// TIA Portal V20 export
TYPE "typeCmInterfaceSoftCam"
// stored: Access Published, Namespace Unit1.Em5
   STRUCT
      ngAndManualInput : "Unit1.Em5.typeCminterfaceSoftCamManualInput";
      magazine : "Unit1.Em5.typeCminterfaceSoftCamMagazine";
   END_STRUCT;
END_TYPE
